// TwinCAT 3 PLC project MainPlc
// Title: MainPlc
// Company: TcOpenGroup
// ProjectVersion: 0.0.0.1
// ProgramVersion: 3.1.4023.0
// libraries:
//   Tc2_Standard, * (Beckhoff Automation GmbH)
//   Tc2_System, * (Beckhoff Automation GmbH)
//   Tc3_Module, * (Beckhoff Automation GmbH)
//   TcoCore, 0.5.0.829 (Vortex.Library)
//   TcoData, 0.5.0.829 (Vortex.Library)
//   TcoInspectors, 0.5.0.829 (Vortex.Library)
//   TcoPneumatics, 0.5.0.829 (Vortex.Library)
// project tree:
//   Abstractions/ CUBaseStatusInfo.TcDUT, CUComponentsBase.TcDUT, CUBase.TcPOU, eCUMode.TcDUT, ICUBase.TcIO, ICUTask.TcIO, TcoInnerTask.TcPOU, TcoTaskedSequencer.TcPOU, TcoTaskedService.TcPOU
//   / MAIN.TcPOU, PlcTask.TcTTO
//   Technology/Data/ EntityHeader.TcDUT, eStations.TcDUT, ProcessData.TcDUT, ProcessDataManager.TcPOU
//   Technology/CU00x/Components/ CU00xComponents.TcDUT
//   Technology/CU00x/ CU00x.TcPOU, CU00xAutomat.TcPOU, CU00xGround.TcPOU, CU00xManual.TcPOU
//   Technology/CU00x/Data/ CU00xProcessData.TcDUT
//   Technology/ Technology.TcPOU
// real-time tasks:
//   TASK PlcTask: cycle T#10ms, priority 20, ADS port 350

CONFIGURATION MainPlc
    RESOURCE PLC ON TwinCAT3
        TASK PlcTask(INTERVAL := T#10ms, PRIORITY := 20);
        PROGRAM MAIN WITH PlcTask : MAIN;
    END_RESOURCE
END_CONFIGURATION

// ---- Abstractions/CUBaseStatusInfo.TcDUT
TYPE
    CUBaseStatusInfo EXTENDS TcoCore.TcoStruct :
    STRUCT
        Mode                   : eCUMode;
        CurrentTaskDescription : STRING;
        CurrentUid             : INT;
        CurrentOperation       : STRING(255);
        CurrentCycleTime       : TIME;
        CurrentIsInStepMode    : BOOL;

    END_STRUCT
END_TYPE

// ---- Abstractions/CUComponentsBase.TcDUT
TYPE
    CUComponentsBase EXTENDS TcoCore.TcoStruct :
    STRUCT
       
    END_STRUCT
END_TYPE

// ---- Abstractions/eCUMode.TcDUT
{attribute 'qualified_only'}
{attribute 'strict'}
TYPE
    eCUMode :
    (
        NoMode         := 0,
        GroundMode     := 10,
        GroundModeDone := 15,
        AutomatMode    := 20,
        ManualMode     := 30
    );
END_TYPE

// ---- Technology/Data/EntityHeader.TcDUT
{attribute wpf [Container(Layout.Stack)]}
{attribute wpf [Group(Layout.Scroll)]}
{attribute addProperty Name "<#Entity header#>"}
TYPE
    EntityHeader EXTENDS TcoCore.TcoStruct :
    STRUCT
        {attribute addProperty Name "<#Reciepe#>"}
        {attribute clr [RenderIgnore("Control", "ShadowControl")]}
        {attribute 'qlik_load:Reciepe'}
        Reciepe : STRING(255);
        {attribute addProperty Name "<#Reciepe created#>"}
        {attribute clr [RenderIgnore("Control", "ShadowControl")]}
        {attribute 'qlik_load:ReciepeCreated'}
        ReciepeCreated : DT;
        {attribute addProperty Name "<#Reciepe modified#>"}
        {attribute clr [RenderIgnore("Control", "ShadowControl")]}
        {attribute 'qlik_load:ReciepeLastModified'}
        ReciepeLastModified : DT;
        {attribute addProperty Name "<#Carrier#>"}
        {attribute clr [RenderIgnore("Control", "ShadowControl")]}
        {attribute 'qlik_load:Carrier'}
        Carrier : STRING;
        {attribute addProperty Name "<#Reset or ground position performed#>"}
        {attribute clr [RenderIgnore("Control", "ShadowControl")]}
        {attribute 'qlik_load:WasReset'}
        {attribute 'qlikmap:Bool:0,No;1,Yes'}
        WasReset : BOOL;
        {attribute addProperty Name "<#Is Master#>"}
        {attribute clr [RenderIgnore("Control", "ShadowControl")]}
        {attribute 'qlik_load:IsMaster'}
        {attribute 'qlikmap:Bool:0,No;1,Yes'}
        IsMaster : BOOL;
        {attribute addProperty Name "<#Is empty#>"}
        {attribute clr [RenderIgnore("Control", "ShadowControl")]}
        {attribute 'qlik_load:IsEmpty'}
        {attribute 'qlikmap:Bool:0,No;1,Yes'}
        IsEmpty : BOOL;
        {attribute addProperty Name "<#Last station#>"}
        {attribute 'qlik_load:LastStation'}
        LastStation : eStations;
        {attribute addProperty Name "<#Next station#>"}
        {attribute 'qlik_load:NextStation'}
        NextStation : eStations;
        {attribute addProperty Name "<#Operations Opened#>"}
        {attribute 'qlik_load:OpenOn'}
        OpenOn : eStations;
        {attribute addProperty Name "<#Results#>"}
        Results : TcoInspectors.TcoComprehensiveResult;

        {attribute addProperty Name "<#Was Reworked#>"}
        {attribute clr [RenderIgnore("Control", "ShadowControl")]}
        {attribute 'qlik_load:WasReworked'}
        WasReworked : BOOL;

        {attribute addProperty Name "<#Last Rework Name#>"}
        {attribute clr [RenderIgnore("Control", "ShadowControl")]}
        {attribute 'qlik_load:LastReworkName'}
        LastReworkName : STRING;

        {attribute addProperty Name "<#Rework Count#>"}
        {attribute clr [RenderIgnore("Control", "ShadowControl")]}
        {attribute 'qlik_load:ReworkCount'}
        ReworkCount : SINT;

    END_STRUCT
END_TYPE

// ---- Technology/Data/eStations.TcDUT
{attribute 'qualified_only'}
{attribute 'strict'}
TYPE
    eStations :
    (
        ST_1  := 1,
        ST_2  := 2,
        ST_3  := 3,
        ST_4  := 4,
        ST_5  := 5,
        ST_6  := 6,
        ST_7  := 7,
        ST_8  := 8,
        ST_9  := 9,
        ST_10 := 10,
        ST_11 := 11,
        ST_12 := 12,
        ST_13 := 13,
        ST_14 := 14,
        ST_15 := 15,
        ST_16 := 16,
        ST_17 := 17,
        ST_18 := 18,
        ST_19 := 19,
        ST_20 := 20,
        NONE  := 32767
    );
END_TYPE

// ---- Technology/Data/ProcessData.TcDUT
{attribute clr [Container(Layout.Tabs)]}
TYPE
    ProcessData EXTENDS TcoData.TcoEntity :
    STRUCT
        {attribute clr [Container(Layout.Stack)]}
        {attribute clr [Group(Layout.GroupBox)]}
        {attribute addProperty Name "<#ID#>"}
        {attribute clr [RenderIgnore()]}
        {attribute 'qlik_association_field'}
        {attribute 'qlik_load:Id'}
        {attribute 'qlik_select:_Id_1'}
        qlikId : STRING(254);
        {attribute clr [RenderIgnore("Control", "ShadowControl")]}
        {attribute addProperty Name "<#Created#>"}
        {attribute 'qlik_time_partition:Shift:[Morning]06:00:00-14:00:00;[Afternoon]14:00:00-22:00:00;[Night]22:00:00-06:00:00'}
        _Created : DT;
        {attribute clr [RenderIgnore("Control", "ShadowControl")]}
        {attribute addProperty Name "<#Modified#>"}
        _Modified : DT;
        {attribute addProperty Name "<#Entity header#>"}
        _entityHeader : EntityHeader     := (Parent := THISSTRUCT);
        CU00x         : CU00xProcessData := (Parent := THISSTRUCT);
    END_STRUCT
END_TYPE

// ---- Technology/CU00x/Components/CU00xComponents.TcDUT
TYPE
    CU00xComponents EXTENDS CUComponentsBase :
    STRUCT
        horizontalCylinder : TcoPneumatics.TcoCylinder(THISSTRUCT);
    END_STRUCT
END_TYPE

// ---- Technology/CU00x/Data/CU00xProcessData.TcDUT
{attribute clr [Container(Layout.Stack)]}
{attribute clr [Group(Layout.Scroll)]}
TYPE
    CU00xProcessData EXTENDS TcoCore.TcoStruct :
    STRUCT
        BoltPresenceInspector : TcoInspectors.TcoDigitalInspector(THISSTRUCT);
    END_STRUCT
END_TYPE

// ---- Abstractions/ICUBase.TcIO
INTERFACE ICUBase

PROPERTY Automat : REFERENCE TO TcoTaskedSequencer
GET
END_GET
END_PROPERTY

PROPERTY Ground : REFERENCE TO TcoTaskedSequencer
GET
END_GET
END_PROPERTY

PROPERTY ProcessDataManager : REFERENCE TO ProcessDataManager
GET
END_GET
END_PROPERTY

END_INTERFACE

// ---- Abstractions/ICUTask.TcIO
INTERFACE ICUTask

PROPERTY Task : REFERENCE TO TcoCore.TcoTask
GET
END_GET
END_PROPERTY

END_INTERFACE

// ---- MAIN.TcPOU
PROGRAM MAIN
VAR
    _technology : Technology;
END_VAR

_technology.Run();

END_PROGRAM

// ---- Technology/Technology.TcPOU
FUNCTION_BLOCK Technology EXTENDS TcoCore.TcoContext
VAR
    _processSettings : ProcessDataManager(THIS^);
    _cu00x           : CU00x(THIS^);
END_VAR

(*~
	<docu>
		<summary>
			Main method of the TcoContext. This is the entry point of any control logic that belongs to this context. 
			The call of this method is ensured by calling the <c>InstanceName.Run()</c> method, and it must not be called explicitly.
			This method is abstract, and it must be overridden in derived block.
		</summary>
	</docu>
~*)
METHOD PROTECTED Main
_cu00x();
END_METHOD

PROPERTY ProcessSettings : REFERENCE TO ProcessDataManager
GET
ProcessSettings REF= _processSettings;
END_GET
END_PROPERTY

METHOD Serve
VAR
	Cu : ICUBase;
END_VAR
END_METHOD

END_FUNCTION_BLOCK

// ---- Technology/Data/ProcessDataManager.TcPOU
FUNCTION_BLOCK ProcessDataManager EXTENDS TcoData.TcoDataExchange
VAR
    _data : ProcessData := (Parent := THIS^);
END_VAR

SUPER^();

PROPERTY Data : REFERENCE TO ProcessData
GET
Data REF= _data;
END_GET
END_PROPERTY

END_FUNCTION_BLOCK

// ---- Technology/CU00x/CU00x.TcPOU
{attribute addProperty ShortName "CU00x"}
{attribute addProperty Name "Controlled unit template"}
FUNCTION_BLOCK CU00x EXTENDS CUBase
VAR
    _cuData      : REFERENCE TO CU00xProcessData;
    _processData : ProcessDataManager(THIS^);
    _components  : CU00xComponents := (Parent := THIS^);
	{attribute addProperty Name "<#AUTOMAT#>"}
	{attribute addProperty ToolTip "<#Starts automatic sequence. Before start you need to perform grounding sequence.#>"}
    _automat     : CU00xAutomat(THIS^, TcoCore.eRestoreMode.None);	
	{attribute addProperty Name "<#GROUND#>"}
	{attribute addProperty ToolTip "<#Brings the device into basic position.#>"}
    _ground      : CU00xGround(THIS^, TcoCore.eRestoreMode.None);
	{attribute addProperty Name "<#MANUAL#>"}
	{attribute addProperty ToolTip "<#Start manual/Service mode#>"}
    _manual      : CU00xManual(THIS^);
END_VAR

_processData();

_automat.Task.Enabled := _ground.GroundDone;
_automat();

_ground.Task.Enabled := NOT _ground.Task.Done;
_ground();

_manual.Task.Enabled := TRUE;
_manual();

UpdateInfo();

PROPERTY Automat : REFERENCE TO TcoTaskedSequencer
GET
Automat REF= _automat;
END_GET
END_PROPERTY

METHOD CancelGround
VAR_INPUT
END_VAR
_ground.CancelGround();
END_METHOD

PROPERTY Components : REFERENCE TO CU00xComponents
GET
Components REF= _components;
END_GET
END_PROPERTY

PROPERTY Ground : REFERENCE TO TcoTaskedSequencer
GET
Ground REF= _ground;
END_GET
END_PROPERTY

METHOD InitializeComponents : BOOL
END_METHOD

PROPERTY Manual : REFERENCE TO TcoTaskedService
GET
Manual REF= _manual;
END_GET
END_PROPERTY

PROPERTY ProcessDataManager : REFERENCE TO ProcessDataManager
GET
ProcessDataManager REF= _processData;
END_GET
END_PROPERTY

PROPERTY Technology : REFERENCE TO Technology
GET
VAR
    _technology : POINTER TO Technology;
END_VAR
IF __QUERYPOINTER(Parent, _technology) THEN // Check if _Parent is Station001
    Technology REF= _technology^;              // If the check is successful dereference a pointer. simlar to THIS^ or SUPER^
END_IF
END_GET
END_PROPERTY

END_FUNCTION_BLOCK

// ---- Abstractions/CUBase.TcPOU
{attribute addProperty ShortName ""}
FUNCTION_BLOCK ABSTRACT CUBase EXTENDS TcoCore.TcoObject IMPLEMENTS ICuBase
VAR
    _statusInfo : CUBaseStatusInfo := (Parent := THIS^);
END_VAR

PROPERTY ABSTRACT Automat : REFERENCE TO TcoTaskedSequencer
GET
END_GET
END_PROPERTY

PROPERTY ABSTRACT Ground : REFERENCE TO TcoTaskedSequencer
GET
END_GET
END_PROPERTY

PROPERTY ABSTRACT Manual : REFERENCE TO TcoTaskedService
GET
END_GET
END_PROPERTY

PROPERTY ABSTRACT ProcessDataManager : REFERENCE TO ProcessDataManager
GET
END_GET
END_PROPERTY

METHOD UpdateInfo : BOOL
VAR_INPUT
END_VAR
IF Automat.Task.Busy THEN
    _statusInfo.Mode                   := eCUMode.AutomatMode;
    _statusInfo.CurrentTaskDescription := '<#AUTOMAT#>';
    _statusInfo.CurrentCycleTime       := Automat._SequenceElapsedTime;
    _statusInfo.CurrentUid             := Automat.CurrentStep.ID;
    _statusInfo.CurrentOperation       := Automat.CurrentStep.Description;
    _statusInfo.CurrentIsInStepMode    := Automat._modeController._mode = eSequencerMode.StepMode;
ELSIF Ground.Task.Busy THEN
    _statusInfo.Mode := eCUMode.GroundMode;
	_statusInfo.CurrentTaskDescription := '<#GROUND#>';
    _statusInfo.CurrentCycleTime       := Ground._SequenceElapsedTime;
    _statusInfo.CurrentUid             := Ground.CurrentStep.ID;
    _statusInfo.CurrentOperation       := Ground.CurrentStep.Description;
    _statusInfo.CurrentIsInStepMode    := Ground._modeController._mode = eSequencerMode.StepMode;
ELSIF THIS^.Manual.Busy THEN
    _statusInfo.Mode := eCUMode.ManualMode;
	_statusInfo.CurrentTaskDescription := '<#MANUAL#>';
ELSIF THIS^.Ground.Task.Done THEN
	_statusInfo.CurrentTaskDescription := '<#READY TO START#>';
	_statusInfo.Mode := eCUMode.GroundModeDone;
	_statusInfo.CurrentCycleTime       := Ground._SequenceElapsedTime;
    _statusInfo.CurrentUid             := Ground.CurrentStep.ID;
    _statusInfo.CurrentOperation       := Ground.CurrentStep.Description;
    _statusInfo.CurrentIsInStepMode    := Ground._modeController._mode = eSequencerMode.StepMode;
ELSE
    _statusInfo.Mode := eCUMode.NoMode;	
	_statusInfo.CurrentTaskDescription := '<#IDLE#>';
	_statusInfo.CurrentCycleTime       := T#0S;
    _statusInfo.CurrentUid             := 0;
    _statusInfo.CurrentOperation       := '';
    _statusInfo.CurrentIsInStepMode    := FALSE;
END_IF
END_METHOD

END_FUNCTION_BLOCK

// ---- Abstractions/TcoTaskedSequencer.TcPOU
FUNCTION_BLOCK PUBLIC ABSTRACT TcoTaskedSequencer EXTENDS TcoCore.TcoSequencerBase
VAR
	{attribute addProperty Name "|[[1]AttributeName]|"}
	{attribute addProperty ToolTip "|[[1]AttributeToolTip]|"}
    _task : TcoInnerTask(THIS^);
    _o    : TcoCore.TcoSequencerObserver(THIS^);	 	
END_VAR

(*~
	<docu>
		<summary>
			<para>
				Completes the sequencer, and return the sequencer pointer to the first step in the seuqence.
				Method is typically called inside the last step of the sequence.
			</para>
		</summary>			
	</docu>	
~*)
METHOD PROTECTED FINAL CompleteSequence
i_CompleteSequence();
END_METHOD

(*~
	<docu>
		<summary>
			Completes the execution of the current step and moves the sequencer pointer to the next step in order of execution.
			The call returns `ITcoObjectRestorer` that allows to restore object upon step completition.
		</summary>		
		<returns></returns>	
	</docu>	
~*)
METHOD PROTECTED FINAL CompleteStep : ITcoObjectRestorer
CompleteStep := i_CompleteStep();
END_METHOD

(*~
	<docu>
		<summary>
			Main method of the sequener. Custom code needs to be placed here. The sequencer is executed by call of **Instance.Run()** method.
			This method is abstract, and it must be overridden in derived block.
		</summary>
	</docu>
~*)
METHOD PROTECTED ABSTRACT Main : BOOL
END_METHOD

METHOD PUBLIC OnAbort : BOOL
END_METHOD

METHOD PUBLIC OnDone : BOOL
END_METHOD

METHOD PUBLIC OnError : BOOL
END_METHOD

METHOD PUBLIC OnStart
END_METHOD

METHOD pr_Close
VAR_INPUT
END_VAR
_lastClosingCycle := Context.StartCycleCount;

IF _sequencerHasError THEN
    OnSequencerError(_sequencerErrorId);
END_IF

_previousNumberOfStepsInSequence := _numberOfStepsInSequence;
Context.Environment.Messaging.Suspend();

IF _modeController._stepIn.Done THEN
    _modeController._stepIn.Restore();
END_IF

Context.Environment.Messaging.Resume();

_restoringSequence := FALSE;
END_METHOD

METHOD pr_Open
VAR
    _message : STRING(255);
END_VAR
_theOrderOfTheCurrentlyEvaluatedStep := 0;

IF _requestStepActive AND
    _requestedStepId <> (MinStepID - 1) AND
    (_modeController.Mode <> eSequencerMode.StepMode OR _modeController._stepIn.Busy OR _checkStepIdRequestedInStepMode) THEN
    _requestStepCycle := _requestStepCycle + 1;
ELSE
    _requestStepCycle := 0;
END_IF

IF _requestStepCycle > 1 AND NOT _sequencerHasError THEN
    _sequencerErrorId        := eSequencerError.StepWithRequestedIdDoesNotExists;
    _message                 := CONCAT('REQUESTED STEP_ID: ', INT_TO_STRING(_requestedStepId));
    _message                 := CONCAT(_message, ' DOES NOT EXIST');
    _currentStep.Description := _message;
    _currentStep.Status      := eStepStatus.Error;
    THIS^.Messenger.Post(_message, eMessageCategory.ProgrammingError);
    _sequencerHasError := TRUE;
END_IF

IF _StepIdUniquenessControlState = eStepIdUniquenessControlState.NotYetStarted OR
    _StepIdUniquenessControlState = eStepIdUniquenessControlState.Requested THEN
    _StepIdUniquenessControlState := eStepIdUniquenessControlState.Started;
END_IF;

_restoringSequence := FALSE;

_lastOpeningCycle := Context.StartCycleCount;
;
END_METHOD

(*~
	<docu>
		<summary>
			Terminates the currently executed step and set the sequencer's pointer to the step with Id that corresponds to ```inRequestedStepID``` parameter.
			When the order of the requested step is higher than the order of the currently finished step (the requested step is "after" the current one)
			the requested step is started in the same context cycle.
			When the order of the requested step is lower than the order of the currently finished step (the requested step is "before" the current one)
			the requested step is started in the next context cycle.
			If the requested step is not found even in the next context cycle, the sequencer enters error state ```StepWithRequestedIdDoesNotExists```.
			<para>
				See <see cref="TcoCore.eSequencerError"/> for detailed description.
			</para>
		</summary>
	</docu>
~*)
METHOD PROTECTED FINAL RequestStep : ITcoSequencer
VAR_INPUT
    (*~
		<docu>
			<summary>
				StepId of the step to be executed.
			</summary>
		</docu>
	~*)
    inRequestedStepID : INT := MinStepID - 1;
END_VAR
VAR
    _message : STRING(254);
END_VAR
RequestStep := i_RequestStep(inRequestedStepID := inRequestedStepID);
END_METHOD

(*~
	<docu>
		<summary>
			<para>
				This method resets the sequencer. 
				Method is typically called before starting the sequence or after error has occured in the sequence.
			</para>
		</summary>			
	</docu>	
~*)
METHOD PUBLIC Restore : ITcoRestorable
SUPER^.Restore();
Task.Restore();
END_METHOD

(*~
	<docu>
		<summary>
			<para>
				Ensures calling the Open(), Main() and Close() methods in the desired order.
				This method is final, so it cannot be overloaded. The **Instance.Run()** needs to be called cyclically inside the appropriate context.
			</para>
		</summary>			
	</docu>	
~*)
METHOD PUBLIC FINAL Run
VAR
    _message : STRING;
END_VAR
IF (_task.Execute()) THEN
    THIS^.pr_Open();
    THIS^.Observer := _o;
    THIS^.Main();
    THIS^.pr_Close();
END_IF;
END_METHOD

METHOD PROTECTED Step : BOOL
VAR_INPUT
    (*~
	<docu>
		<summary>
			StepId of the current step.
			<remarks>			
				<note type="important">
					This number must be unique throughout the complete sequence.
					It must be a constant or numerical literal and it must not change during the life-time of the sequencer. 
				</note>
			</remarks>
		</summary>		
	</docu>	
~*)
    inStepID : INT;
    (*~
	<docu>
		<summary>
			If this value is false, step body is not executed and execution is moved to the next enabled step.
		</summary>				
	</docu>	
~*)
    inEnabled : BOOL;
    (*~
	<docu>
		<summary>
			Step description text.
		</summary>				
	</docu>	
~*)
    inStepDescription : STRING(254);
END_VAR
Step := i_Step(inStepID := inStepID, inEnabled := inEnabled, inStepDescription := inStepDescription);
END_METHOD

(*~
	<docu>
		<summary>
			Completes the actually running step, when the `inCondition` parameter is `TRUE`.
			Method is typically called inside a step as the transition method.
		</summary>			
	</docu>	
~*)
METHOD PROTECTED FINAL StepCompleteWhen
VAR_INPUT
    (*~
	<docu>
		<summary>
			The condition under which the step is completed.
		</summary>			
	</docu>	
~*)
    inCondition : BOOL;
END_VAR
i_StepCompleteWhen(inCondition := inCondition);
END_METHOD

PROPERTY Task : REFERENCE TO TcoTask
GET
Task REF= _task;
END_GET
END_PROPERTY

END_FUNCTION_BLOCK

// ---- Abstractions/TcoInnerTask.TcPOU
FUNCTION_BLOCK TcoInnerTask EXTENDS TcoCore.TcoTask

(*~
	<docu>
		<summary>
			Executes when task is aborted.
		</summary>			
	</docu>	
~*)
METHOD PROTECTED OnAbort
ParentSequencer.OnAbort();
END_METHOD

(*~
	<docu>
		<summary>
			Executes when task reaches the ```Done``` state .
		</summary>			
	</docu>	
~*)
METHOD PROTECTED OnDone
ParentSequencer.OnDone();
END_METHOD

(*~
	<docu>
		<summary>
			Executes when task reaches the ```Error``` state.
			<para>
				Do not confuse with <see cref="PlcDocu.TcoCore.TcoTask.WhileError()"/>, that is called cyclically until '''Error''' state is left.
			</para>
		</summary>			
	</docu>	
~*)
METHOD PROTECTED OnError
ParentSequencer.OnError();
END_METHOD

METHOD PROTECTED OnStart
ParentSequencer.OnStart();
END_METHOD

PROPERTY PRIVATE ParentSequencer : REFERENCE TO TcoTaskedSequencer
GET
VAR
	_sequencer : POINTER TO TcoTaskedSequencer;
END_VAR
IF __QUERYPOINTER(Parent, _sequencer) THEN // Check if _Parent is Station001
    ParentSequencer REF= _sequencer^;              // If the check is successful dereference a pointer. simlar to THIS^ or SUPER^
END_IF
END_GET
END_PROPERTY

END_FUNCTION_BLOCK

// ---- Abstractions/TcoTaskedService.TcPOU
FUNCTION_BLOCK PUBLIC ABSTRACT TcoTaskedService EXTENDS TcoCore.TcoTask
VAR
	
END_VAR

(*~
	<docu>
		<summary>
			Main method of the sequener. Custom code needs to be placed here. The sequencer is executed by call of **Instance.Run()** method.
			This method is abstract, and it must be overridden in derived block.
		</summary>
	</docu>
~*)
METHOD PROTECTED ABSTRACT Main : BOOL
END_METHOD

(*~
	<docu>
		<summary>
			<para>
				Ensures calling the Open(), Main() and Close() methods in the desired order.
				This method is final, so it cannot be overloaded. The **Instance.Run()** needs to be called cyclically inside the appropriate context.
			</para>
		</summary>			
	</docu>	
~*)
METHOD PUBLIC FINAL Run
VAR
    _message : STRING;
END_VAR
IF (THIS^.Execute()) THEN
    THIS^.Main();    
END_IF;
END_METHOD

PROPERTY Task : REFERENCE TO TcoTask
GET
Task REF= THIS^;
END_GET
END_PROPERTY

END_FUNCTION_BLOCK

// ---- Technology/CU00x/CU00xAutomat.TcPOU
FUNCTION_BLOCK CU00xAutomat EXTENDS TcoTaskedSequencer IMPLEMENTS ICUTask
VAR
END_VAR

Run();

(*~
	<docu>
		<summary>
			Main method of the sequener. Custom code needs to be placed here. The sequencer is executed by call of **Instance.Run()** method.
			This method is abstract, and it must be overridden in derived block.
		</summary>
	</docu>
~*)
METHOD PROTECTED Main : BOOL
IF (Step(100, TRUE, 'LOAD PROCESS SETTING')) THEN
    //-------------------------------------
    Station.ProcessDataManager.Data := Station.Technology.ProcessSettings.Data;
	CompleteStep();
    //-------------------------------------
END_IF

IF (Step(200, TRUE, 'SINGLE INSPECTION')) THEN
    //-------------------------------------    
	Station.ProcessDataManager.Data.CU00x.BoltPresenceInspector
					.WithCoordinator(THIS^)
					.Inspect(FALSE)
					.UpdateComprehensiveResult(Station.ProcessDataManager.Data._entityHeader.Results)
					.OnFail().Dialog(100);	
    //-------------------------------------
END_IF

IF (Step(RESTORE_STEP_ID, TRUE, 'FIRST RESTORE STEP')) THEN
    //-------------------------------------
    StepCompleteWhen(%MX0.0);
    //-------------------------------------	
END_IF

IF (Step(10000, TRUE, 'LAST STEP')) THEN
    //-------------------------------------
    CompleteSequence();
    //-------------------------------------	
END_IF
END_METHOD

METHOD PUBLIC OnStart
Station.Ground.Restore();
Station.Manual.Restore();
END_METHOD

PROPERTY Station : REFERENCE TO CU00x
GET
VAR
    _station : POINTER TO CU00x;
END_VAR
IF __QUERYPOINTER(Parent, _station) THEN // Check if _Parent is Station001
    Station REF= _station^;              // If the check is successful dereference a pointer. simlar to THIS^ or SUPER^
END_IF
END_GET
END_PROPERTY

END_FUNCTION_BLOCK

// ---- Technology/CU00x/CU00xGround.TcPOU
FUNCTION_BLOCK CU00xGround EXTENDS TcoTaskedSequencer IMPLEMENTS ICUTask
VAR
	_groundDone : BOOL;
END_VAR

Run();

METHOD CancelGround
_groundDone := FALSE;
END_METHOD

PROPERTY GroundDone : BOOL
GET
GroundDone := _groundDone;
END_GET
END_PROPERTY

(*~
	<docu>
		<summary>
			Main method of the sequener. Custom code needs to be placed here. The sequencer is executed by call of **Instance.Run()** method.
			This method is abstract, and it must be overridden in derived block.
		</summary>
	</docu>
~*)
METHOD PROTECTED Main : BOOL
IF (Step(100, TRUE, 'STOPPING OTHER MODES')) THEN
	Station.Automat.Restore();
	Station.Manual.Restore();
    CompleteStep();
END_IF

IF (Step(200, TRUE, 'STOPPING OTHER MODES')) THEN	
    StepCompleteWhen(THIS^._currentStep.Duration > T#3S);
END_IF

IF (Step(10000, TRUE, 'LAST STEP')) THEN	
	_groundDone := TRUE;
	THIS^._task.DoneWhen(_groundDone);
END_IF
END_METHOD

METHOD PUBLIC OnStart
Station.Automat.Restore();
Station.Manual.Restore();
END_METHOD

PROPERTY Station : REFERENCE TO CU00x
GET
VAR
    _station : POINTER TO CU00x;
END_VAR
IF __QUERYPOINTER(Parent, _station) THEN // Check if _Parent is Station001
    Station REF= _station^;              // If the check is successful dereference a pointer. simlar to THIS^ or SUPER^
END_IF
END_GET
END_PROPERTY

END_FUNCTION_BLOCK

// ---- Technology/CU00x/CU00xManual.TcPOU
FUNCTION_BLOCK CU00xManual EXTENDS TcoTaskedService IMPLEMENTS ICUTask
VAR
END_VAR

Run();

(*~
	<docu>
		<summary>
			Main method of the sequener. Custom code needs to be placed here. The sequencer is executed by call of **Instance.Run()** method.
			This method is abstract, and it must be overridden in derived block.
		</summary>
	</docu>
~*)
METHOD PROTECTED Main : BOOL
Station.Components.horizontalCylinder.Service();
END_METHOD

METHOD PROTECTED OnStart
Station.Automat.Restore();
Station.Ground.Restore();
Station.CancelGround();
END_METHOD

PROPERTY Station : REFERENCE TO CU00x
GET
VAR
    _station : POINTER TO CU00x;
END_VAR
IF __QUERYPOINTER(Parent, _station) THEN // Check if _Parent is Station001
    Station REF= _station^;              // If the check is successful dereference a pointer. simlar to THIS^ or SUPER^
END_IF
END_GET
END_PROPERTY

END_FUNCTION_BLOCK
